KUKA KRL data list: ui_helper.dat

&ACCESS RV1
DEFDAT  ui_helper PUBLIC

ENDDAT
